FUNCTION_BLOCK BUTTONChan (* Composite Function Block Type *)
  (* Standard: 61499-2 *)
  (* Version 0.0, 7/20/2013, vvya002, nxtControl GmbH, template *)
  PACKAGE Main;
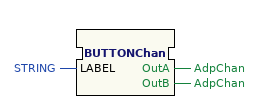
  VAR_INPUT
    LABEL : STRING;
  END_VAR
  PLUGS
    OutA : AdpChan;
    OutB : AdpChan;
  END_PLUGS
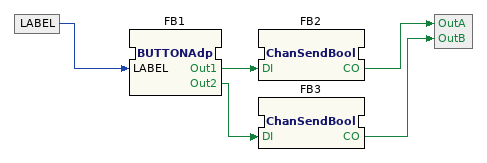
  FBS
    FB1 : BUTTONAdp;
    FB2 : ChanSendBool;
    FB3 : ChanSendBool;
  END_FBS
  DATA_CONNECTIONS
    LABEL TO FB1.LABEL;
  END_CONNECTIONS
  ADAPTER_CONNECTIONS
    FB1.Out1 TO FB2.DI;
    FB1.Out2 TO FB3.DI;
    FB2.CO TO OutA;
    FB3.CO TO OutB;
  END_CONNECTIONS
END_FUNCTION_BLOCK
